(* PLC project Proj1, Beckhoff Automation GmbH TwinCAT PLC Control 3.5.20.60 *)
(* stored: creationDateTime 2025-10-20T07:57:40.286671, modificationDateTime 2025-10-20T07:57:40.2956466 *)

FUNCTION_BLOCK PUBLIC FB_Automatikbetrieb_F1
VAR_INPUT
    Automatikbetrieb_Starten : BOOL;
	AutoRestartEnable   : BOOL;      // Schalter für Autorestart
    // <<< NEU: parametrierbarer, periodischer Störgenerator >>>
    PeriodicFaultEnable : BOOL := TRUE;       // Ein/Aus
    PeriodicFaultPeriod : TIME := T#60s;      // z. B. jede Minute
    FaultPulse          : TIME := T#100ms;    // wie lange „Störung“ getriggert wird
END_VAR
VAR RETAIN
    lastSkillIsOne : BOOL := FALSE; // FALSE => erster Start wird TestSkill3 -> wir setzen gleich initial um
END_VAR
VAR_OUTPUT
    Automatikbetrieb_Fertig : BOOL;
    Stoerung_erkannt        : BOOL;
END_VAR
VAR
    Schritt1 : BOOL;
    Schritt2 : BOOL;
	Zwischen : STRING;
    tSchritt1 : TON;
    tSchritt2 : TON;
    rStart   : R_TRIG;
    rtStoer   : R_TRIG;
	rStep1 : R_TRIG;

    // <<< NEU >>>
    tPer   : TON;      // Periodentimer
    rPer   : R_TRIG;   // Flanke bei Periodenende
    pPer   : TP;       // kurzer Puls für die Störung
    perEn  : BOOL;     // Enable nur wenn die Automatik läuft
    dbg_Stoerung_Manuell : BOOL; // hattest du schon
	tpRestart: INT;
	RestartPulseLength: INT;
END_VAR

                  
//GVL.Start := TRUE;
IF GVL.Start THEN
	AutoRestartEnable := TRUE;
END_IF
// === Flanken bilden ===
rStart(CLK := Automatikbetrieb_Starten);
rStep1(CLK := Schritt1);

// === Startsequenz auf positive Flanke, nur wenn nicht bereits aktiv ===
IF (AutoRestartEnable AND NOT (Schritt1 OR Schritt2)) OR (Stoerung_erkannt AND GVL.Weiter) THEN
    // Reset aller Zustände
    Automatikbetrieb_Fertig := FALSE;
    Stoerung_erkannt        := FALSE;
	GVL.Weiter := FALSE;
    // Start in Schritt 1
    Schritt1 := TRUE;
	OPCUA.lastExecutedProcess := 'ExTechnProcess1';
    Schritt2 := FALSE;
END_IF

// === Timer an die Schritte koppeln ===
tSchritt1(IN := Schritt1, PT := T#55S);
tSchritt2(IN := Schritt2, PT := T#55S);

IF rStep1.Q THEN
    lastSkillIsOne := NOT lastSkillIsOne;
    IF lastSkillIsOne THEN
        OPCUA.lastExecutedSkill := 'TestSkill1';
    ELSE
        OPCUA.lastExecutedSkill := 'TestSkill1';
    END_IF
END_IF

IF rStart.Q AND NOT (Schritt1 OR Schritt2) THEN
    Automatikbetrieb_Fertig := FALSE;
    Stoerung_erkannt := FALSE;
    GVL.Weiter := FALSE;
    Schritt1 := TRUE;
    Schritt2 := FALSE;
    OPCUA.lastExecutedProcess := 'ExTechnProcess1';
END_IF

// === Übergänge (sofern keine Störung aktiv ist) ===
IF NOT Stoerung_erkannt THEN
    // Schritt 1 -> 2 nach 30 s
    IF Schritt1 AND tSchritt1.Q THEN
        Schritt1 := FALSE;
        Schritt2 := TRUE;
		OPCUA.lastExecutedSkill := 'TestSkill1';
    END_IF

    // Schritt 2 -> Fertig nach 10 s
    IF Schritt2 AND tSchritt2.Q THEN
        Schritt2 := FALSE;
        Automatikbetrieb_Fertig := TRUE;
        // Hier KEIN automatischer Neustart; neuer Start benötigt erneute Startflanke
    END_IF
END_IF

// === Störungen behandeln (manuell) ===
IF rtStoer.Q THEN
    Stoerung_erkannt := TRUE;
END_IF

/// frei laufender Periodentimer (unabhängig von Schritt1/2) für Störung
tPer(IN := NOT tPer.Q, PT := PeriodicFaultPeriod);  // z.B. T#60s

// Flanke bei Periodenende + definierter Puls
rPer(CLK := tPer.Q);
pPer(IN := rPer.Q, PT := FaultPulse);                // z.B. T#100ms

// nur auslösen, wenn die Automatik gerade läuft
IF (Schritt1 OR Schritt2) AND pPer.Q THEN
    Stoerung_erkannt := TRUE;
	GVL.Fehler := TRUE;
END_IF


                
END_FUNCTION_BLOCK

FUNCTION_BLOCK FB_Betriebsarten
VAR_INPUT
	Start, NotStop, Weiter, Fehler, Start_Init : BOOL;
    Auto_Fertig   : BOOL; // kommt von fbAuto.Automatikbetrieb_Fertig
    Auto_Stoerung : BOOL; // kommt von fbAuto.Stoerung_erkannt
	A2_Requested: BOOL;
	Alt_abort: BOOL;
	Alt_found: BOOL;
	D3_Requested: BOOL;
	Init_reached: BOOL;
	Cycle_ended: BOOL;
	//Reset			: BOOL;
	//Schalter		: BOOL;
	//Schrittkette_GS : BOOL;
END_VAR
VAR_OUTPUT
	A1 : BOOL; //Initialzustand
	A2 : BOOL; //Stillstand angefordert am Ende des Zyklus
//	A3 : BOOL; //Stillstand angefordert in einem bestimmten Zustand
//	A4 : BOOL; //Erhaltener Stillstand
	A5 : BOOL; //Vorbereitung zur Wiederaufnahme nach Störung
	A6 : BOOL; //Fahrt in den Initialzustand
	F1 : BOOL; //Normalbetrieb
//	F2 : BOOL; //Anfahren
//	F3 : BOOL; //Abfahren
	F4 : BOOL; //Handbetrieb
//	F5 : BOOL; //Schrittbetrieb
//	F6 : BOOL; //Testbetrieb
	D1 : BOOL; //Not-Aus
	D2 : BOOL; //DIagnose und Störbehandlung
	D3 : BOOL; //Produktion trotz Störung
END_VAR
VAR
	bFirstScan : BOOL := TRUE;	

	RS_InitialState: RS;	
	RS_InitialDrive: RS;
	RS_ManualOperationMode: RS;
	RS_AutomaticOperationMode: RS;
	RS_CycleEnded: RS;

	R_TRIG_Manual: R_TRIG;
	R_TRIG_Automatic: R_TRIG;
	R_TRIG_InitialDrive: R_TRIG;
	R_TRIG_CycleEnded: R_TRIG;
	R_TRIG_Init: R_TRIG;
	RS_D2: RS;
	RS_F1: RS;
	RS_D1: RS;
	RS_A5: RS;
	RS_A1: RS;

	RS_D3: RS;

	RS_A2: RS;
	RS_A6: RS;
END_VAR

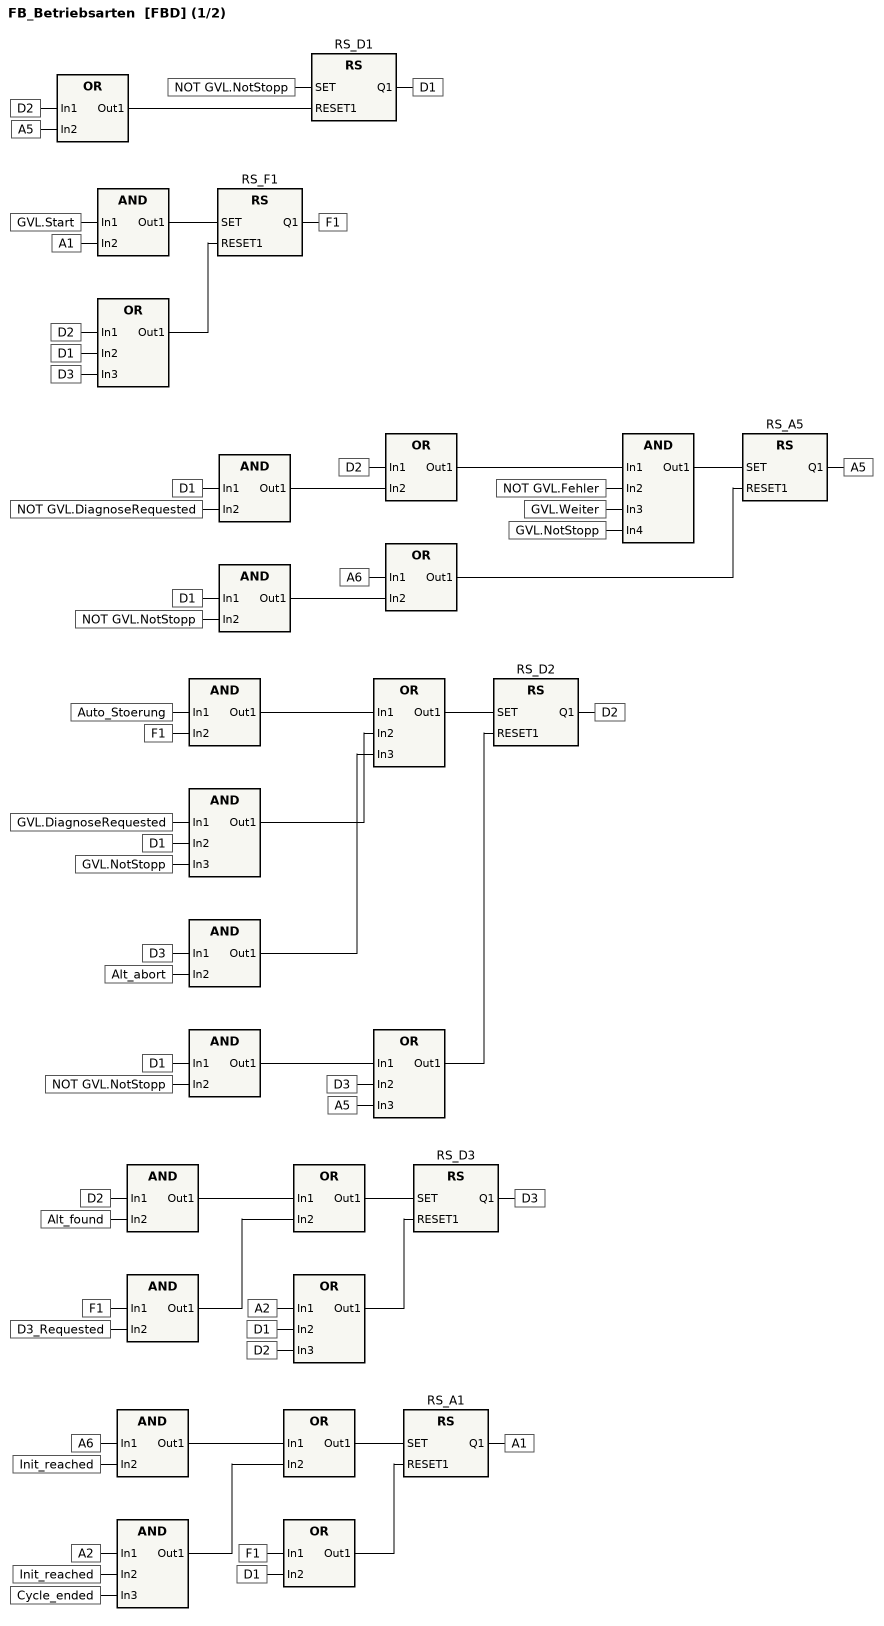
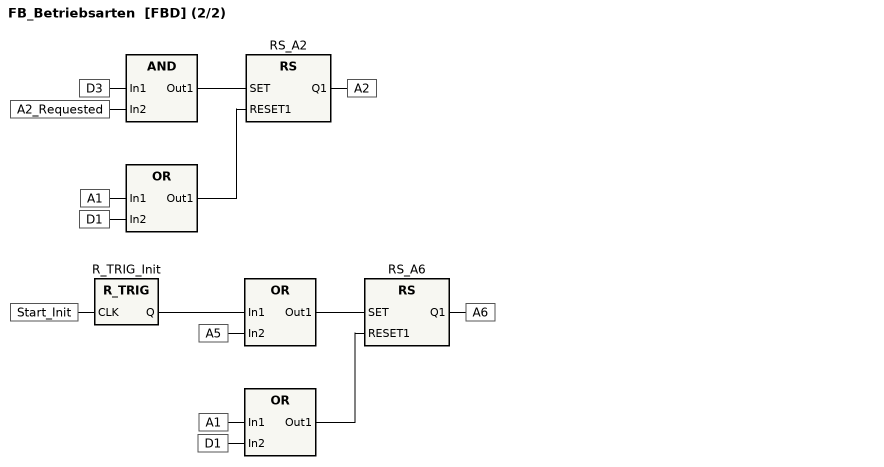
(* FBD diagram, written out as Structured Text *)
RS_D1(SET := NOT GVL.NotStopp, RESET1 := D2 OR A5);
D1 := RS_D1.Q1;
RS_F1(SET := GVL.Start AND A1, RESET1 := D2 OR D1 OR D3);
F1 := RS_F1.Q1;
RS_A5(SET := (D2 OR D1 AND (NOT GVL.DiagnoseRequested)) AND (NOT GVL.Fehler) AND GVL.Weiter AND GVL.NotStopp, RESET1 := A6 OR D1 AND (NOT GVL.NotStopp));
A5 := RS_A5.Q1;
RS_D2(SET := Auto_Stoerung AND F1 OR GVL.DiagnoseRequested AND D1 AND GVL.NotStopp OR D3 AND Alt_abort, RESET1 := D1 AND (NOT GVL.NotStopp) OR D3 OR A5);
D2 := RS_D2.Q1;
RS_D3(SET := D2 AND Alt_found OR F1 AND D3_Requested, RESET1 := A2 OR D1 OR D2);
D3 := RS_D3.Q1;
RS_A1(SET := A6 AND Init_reached OR A2 AND Init_reached AND Cycle_ended, RESET1 := F1 OR D1);
A1 := RS_A1.Q1;
RS_A2(SET := D3 AND A2_Requested, RESET1 := A1 OR D1);
A2 := RS_A2.Q1;
R_TRIG_Init(CLK := Start_Init);
RS_A6(SET := R_TRIG_Init.Q OR A5, RESET1 := A1 OR D1);
A6 := RS_A6.Q1;
END_FUNCTION_BLOCK

FUNCTION_BLOCK PUBLIC FB_Diagnose_D2
VAR_INPUT
    Diagnose_gefordert         : BOOL;  // z. B. D2 aus FB_Betriebsarten
END_VAR
VAR_OUTPUT
    Diagnose_beendet           : BOOL;  // geht zurück an FB_Betriebsarten
	Alt_gefunden			   : BOOL := FALSE;
END_VAR
VAR
    // Steuerung/Handshake intern
    Busy       : BOOL;

    // Flanken + Puls
    rtReq      : R_TRIG;    // steigende Flanke auf Diagnose_gefordert
	rtD3 : R_TRIG;
    tpPulse    : TP;        // kurzer Puls für OPCUA.TriggerD2 (z. B. 100 ms)
    rtFinished : R_TRIG;    // steigende Flanke auf OPCUA.DiagnoseFinished
	 rtAck : R_TRIG;
END_VAR

                  // 1) Startflanke erkennen
rtReq(CLK := Diagnose_gefordert);

// 2) Einmalig triggern (nur wenn noch nicht "Busy"):
IF rtReq.Q AND NOT Busy THEN
    Busy := TRUE;
	Alt_gefunden := FALSE;
	OPCUA.TriggerD2 := TRUE; 
	OPCUA.bool1 := TRUE;
END_IF

  // {attribute 'OPC.UA.DA' := '1'} in der GVL setzen

// 3) Fertigmeldung vom OPC-UA-Client
//rtFinished(CLK := OPCUA.DiagnoseFinished);
rtAck(CLK := OPCUA.DiagnoseFinished);
rtD3(CLK := OPCUA.Alt_found);
IF rtAck.Q OR rtD3.Q THEN
    Diagnose_beendet := TRUE;
    GVL.Weiter := TRUE;
    Busy := FALSE;
    OPCUA.TriggerD2 := FALSE;
	OPCUA.bool2 := FALSE;
    GVL.Fehler := FALSE;
    Diagnose_gefordert := FALSE;
	GVL.DiagnoseRequested := FALSE;
END_IF
IF rtD3.Q THEN
	Alt_gefunden := TRUE;
END_IF
                
END_FUNCTION_BLOCK

FUNCTION_BLOCK FB_InitFahrt_A6_A2
VAR_INPUT
	A6 : BOOL := FALSE;
	A2: BOOL := FALSE;
END_VAR
VAR_OUTPUT
	Init_erreicht : BOOL := FALSE;
END_VAR
VAR
	tInit : TON;
END_VAR

                  IF A6 THEN
	tInit(IN := A6, PT := T#3S);
ELSIF A2 THEN
	tInit(IN := A2, PT := T#5S);
END_IF

IF tInit.Q THEN
	Init_erreicht := TRUE;
ELSE
	Init_erreicht := FALSE;
END_IF
                
END_FUNCTION_BLOCK

FUNCTION_BLOCK FB_ProduktionMitStoerung_D3
VAR_INPUT
    ProduktionMitStoerung_Starten : BOOL;
END_VAR
VAR RETAIN
    lastSkillIsOne : BOOL := FALSE; // FALSE => erster Start wird TestSkill3 -> wir setzen gleich initial um
END_VAR
VAR_OUTPUT
    Fertig : BOOL;
    Stoerung_erkannt        : BOOL;
END_VAR
VAR
    Schritt3 : BOOL;
    Schritt4 : BOOL;
	Zwischen : STRING;
    tSchritt3 : TON;
    tSchritt4 : TON;
    rStart   : R_TRIG;
    rtStoer   : R_TRIG;
	rStep1 : R_TRIG;
	z : INT := 0;

    // <<< NEU >>>
    tPer   : TON;      // Periodentimer
    rPer   : R_TRIG;   // Flanke bei Periodenende
    pPer   : TP;       // kurzer Puls für die Störung
    perEn  : BOOL;     // Enable nur wenn die Automatik läuft
    dbg_Stoerung_Manuell : BOOL; // hattest du schon
	tpRestart: INT;
	RestartPulseLength: INT;
END_VAR

                  rStart(CLK := ProduktionMitStoerung_Starten);
IF rStart.Q THEN
	z := 0;
END_IF

IF ProduktionMitStoerung_Starten AND NOT (Schritt3 OR Schritt4) AND NOT Stoerung_erkannt THEN
	Fertig := FALSE;
	Schritt3 := TRUE;
	OPCUA.lastExecutedSkill := 'TestSkill3';
	OPCUA.lastExecutedProcess := 'D3Process';
	Schritt4 := FALSE;
END_IF

tSchritt3(IN := Schritt3, PT:=T#10S);
tSchritt4(IN := Schritt4, PT:=T#10S);

IF tSchritt3.Q THEN
	Schritt3 := FALSE;
	z := z+1;
	IF z > 2 THEN
		Stoerung_erkannt := TRUE;
		OPCUA.Alt_abort := TRUE;
	END_IF
	IF NOT Stoerung_erkannt THEN
		Schritt4 := TRUE;
		OPCUA.lastExecutedSkill := 'TestSkill4';
	END_IF
END_IF

IF tSchritt4.Q THEN
	Schritt4 := FALSE;
	Schritt3 := TRUE;
	OPCUA.lastExecutedSkill := 'TestSkill3';
END_IF




                
END_FUNCTION_BLOCK

PROGRAM MAIN
VAR
	{attribute 'OPC.UA.DA' := '1'}       // falls Server im Filter-/Symbolmodus
    fbJob : FB_Methode1Job;              // FB mit {attribute 'OPC.UA.DA.JobMethod' := 'M_Methode1'}
    fbBA   : FB_Betriebsarten;
    fbAuto : FB_Automatikbetrieb_F1;
    fbDiag : FB_Diagnose_D2;
	fbNot : FB_Notaus_D1;
	fbInit : FB_InitFahrt_A6_A2;
	fbProStoer : FB_ProduktionMitStoerung_D3;
	
	Init_start : BOOL := TRUE;
	

    edgeF1    : R_TRIG;  // F1 -> Start Automatik
    edgeDone  : R_TRIG;  // Diagnose_beendet -> Restart/Weiter
	alt_abort : BOOL := FALSE;
	alt_found : BOOL := FALSE;
    Start_eff  : BOOL := FALSE;
    Weiter_eff : BOOL := FALSE;
	A2_angefordert : BOOL := FALSE;
	D3_angefordert : BOOL := FALSE;
	Init_erreicht : BOOL := FALSE;
	Zyklus_beendet : BOOL := FALSE;
	
END_VAR

                  // Diagnose fertig -> Impuls
edgeDone(CLK := fbDiag.Diagnose_beendet);

// manuell ODER automatisch (Restart nach Diagnose)
Start_eff  := GVL.Start  OR edgeDone.Q;
Weiter_eff := GVL.Weiter OR edgeDone.Q;

// Betriebsarten (RS-F1/RS-D2 sind dort)
fbBA(
    Start         := Start_eff,
    NotStop       := GVL.NotStopp,
    Weiter        := Weiter_eff,
    Fehler        := GVL.Fehler,
	Start_Init 	  := Init_Start,                  
    Auto_Fertig   := fbAuto.Automatikbetrieb_Fertig,
    Auto_Stoerung := fbAuto.Stoerung_erkannt,
	A2_Requested := A2_angefordert,
	Alt_abort := alt_abort,
	Alt_found := alt_found,
	D3_Requested := D3_angefordert,
	Init_reached := Init_erreicht,
	Cycle_ended := Zyklus_beendet
);

// F1-Flanke startet die Automatik
edgeF1(CLK := fbBA.F1);
fbAuto(Automatikbetrieb_Starten := edgeF1.Q);

fbNot(D1 := fbBA.D1);
GVL.DiagnoseRequested := fbNot.Diagnose_gefordert;

fbProStoer(ProduktionMitStoerung_Starten := fbBA.D3);
alt_abort := fbProStoer.Stoerung_erkannt;


fbInit(A6 := fbBA.A6, A2 := fbBA.A2);
Init_erreicht := fbInit.Init_erreicht;

// D2 fordert die Diagnose an
fbDiag(Diagnose_gefordert := fbBA.D2);
alt_found := fbDiag.Alt_gefunden;
                
END_PROGRAM

{attribute 'OPC.UA.DA.JobMethod' := 'M_Methode1'} // Dieser FB wird als OPC-UA-Job "M_Methode1" veröffentlicht
FUNCTION_BLOCK FB_Methode1Job
VAR
    running : BOOL := FALSE;
    counter : DINT := 0;
    reached : BOOL := FALSE;
    t20s    : TON;        // 20-s-Timer, läuft zyklisch
    y       : DINT := 0;  // Ergebnis
END_VAR
// Wichtig: Bei Job-Methoden deklariert man den Funktionsbaustein mit
//{attribute 'OPC.UA.DA.JobMethod' := 'NameDerUAMethod'}
//und markiert die drei PLC-METHODs Start, CheckState, Abort jeweils mit TcRpcEnable. 
//CheckState besitzt zwingend das Output bBusy, über das der Server erkennt, ob der Job noch läuft.

                  
                

{attribute 'TcRpcEnable' := '1'}
METHOD PUBLIC Abort : HRESULT
// Aufräumen bei Server-Shutdown/Abbruch
                        running := FALSE;
Abort := 0;
                      
END_METHOD

{attribute 'TcRpcEnable' := '1'}
METHOD PUBLIC CheckState : HRESULT
VAR_INPUT
    hdl : UDINT;       // vom Server übergeben (wenn genutzt)
END_VAR
VAR_OUTPUT
    bBusy : BOOL;      // **erforderlich** für Job-Methode
    yOut  : DINT;      // UA-Output
END_VAR
                        // Mehrzyklische Job-Logik:
IF running THEN
	
    //counter := counter + 1;
    //IF counter >= 30 THEN
        //reached := TRUE;
    //END_IF; 
	reached := TRUE;

    // Timer startet erst ab "reached"
    t20s(IN := reached, PT := T#9S);

    IF reached AND t20s.Q THEN
        y := 119;
        running := FALSE;
    END_IF
END_IF

bBusy := running;
yOut  := y;
CheckState := 0;       // 0 = Good (bei Fehler z. B. BadOutOfRange als HRESULT zurückgeben)
                      
END_METHOD

{attribute 'TcRpcEnable' := '1'}
METHOD PUBLIC Start : HRESULT
VAR_INPUT
    x : DINT;           // Eingabe der UA-Methode
END_VAR
VAR_OUTPUT
    hdl : UDINT;        // optionaler Handle für parallele Aufrufe
END_VAR
                        // Initialisierung
counter := x;
reached := FALSE;
running := TRUE;
t20s(IN := FALSE, PT := T#9S);   // Timer Reset
hdl := 0;                         // (einfacher Fall)
Start := 0;                       // 0 = OPC UA StatusCode "Good"
                      
END_METHOD
END_FUNCTION_BLOCK

FUNCTION_BLOCK FB_Notaus_D1
VAR_INPUT
	D1 : BOOL;
END_VAR
VAR_OUTPUT
	Notaus_Entriegelt : BOOL;
	Diagnose_gefordert : BOOL;
END_VAR
VAR
	ton5s : TON;
END_VAR

                  IF D1 THEN
    OPCUA.TriggerD1 := TRUE;         // interne publizierte Variable (kein AT %I*)
    ton5s(IN := TRUE, PT := T#5S);
ELSE
    ton5s(IN := FALSE, PT := T#5S);
END_IF;

IF ton5s.Q THEN
    OPCUA.TriggerD1 := FALSE;
    Diagnose_gefordert := FALSE;
    GVL.NotStopp := TRUE;
    GVL.Fehler := FALSE;
    GVL.Weiter := TRUE;
END_IF;
                
END_FUNCTION_BLOCK

CONFIGURATION Application
  RESOURCE Proj1 ON PLC
(* global variable list GVL *)
{attribute 'qualified_only'}
VAR_GLOBAL
	Start : BOOL;
	Stopp : BOOL := FALSE;
	NotStopp : BOOL := TRUE;
	Fehler			: BOOL;
	Weiter			: BOOL;
	DiagnoseRequested: BOOL;
END_VAR
(* global variable list OPCUA *)
{attribute 'qualified_only'}
VAR_GLOBAL
	
	{attribute 'OPC.UA.DA' := '1'}
	bool1: BOOL := FALSE;
	{attribute 'OPC.UA.DA' := '1'}
	bool2: BOOL := FALSE;
	{attribute 'OPC.UA.DA' := '1'}
	bool3: BOOL := FALSE;
	
	{attribute 'OPC.UA.DA' := '1'}
	Z1: INT := 0;
	{attribute 'OPC.UA.DA' := '1'}
	Z2: INT := 0;
	{attribute 'OPC.UA.DA' := '1'}
	Z3: INT := 0;
	{attribute 'OPC.UA.DA' := '1'}
    TriggerD2: BOOL := FALSE;
	{attribute 'OPC.UA.DA' := '1'}
    TriggerD1: BOOL := FALSE;
	{attribute 'OPC.UA.DA' := '1'}
    TriggerD3: BOOL := FALSE;
	{attribute 'OPC.UA.DA' := '1'}
    lastExecutedSkill: STRING := '';
	{attribute 'OPC.UA.DA' := '1'}
    lastExecutedProcess: STRING := '';
	{attribute 'OPC.UA.DA' := '1'}
    M1: INT := 0;
	{attribute 'OPC.UA.DA' := '1'}
	M2: INT := 0;
	{attribute 'OPC.UA.DA' := '1'}
	M3: INT := 0;
	{attribute 'OPC.UA.DA' := '1'}
	{attribute 'OPC.UA.Access' := 'readwrite'}
	DiagnoseFinished: BOOL := FALSE;
	{attribute 'OPC.UA.DA' := '1'}
	{attribute 'OPC.UA.Access' := 'readwrite'}
	Alt_found: BOOL := FALSE;
	{attribute 'OPC.UA.DA' := '1'}
	{attribute 'OPC.UA.Access' := 'readwrite'}
	Alt_abort : BOOL := FALSE;
	
	
END_VAR
    TASK PlcTask(INTERVAL := T#0ms, PRIORITY := 20);
    PROGRAM MAIN WITH PlcTask : MAIN;
  END_RESOURCE
END_CONFIGURATION
